VAR_GLOBAL
	/// instance array of all controller instances
	g_a_pCtrlInst: ARRAY[0..E_CtrlId.E_CtrlIdMax] OF POINTER TO fb_CtrlBase;
	/// common interface array of all controllers (main use for PLC)
	g_a_pCtrlCIf: ARRAY[0..E_CtrlId.E_CtrlIdMax] OF POINTER TO T_Ctrl_CIf;
	/// common access variabel for UI
	g_p_fbAlm_Man: POINTER TO FB_Alm_Man;
	/// Global array for function with different childs in faster cycles
	g_a_pFunRFD: ARRAY[0..9] OF POINTER TO FB_RFR;
	/// For StartUp order
	g_uinStartProzess: UINT;
	/// Count of Task Classes
	c_uinCntTaskClass: UINT := 3;
END_VAR

(* stored: Version 1.1.0.1, ProductVersion 3.1.0.23
   GVL Global: Id {c27aced4-be9c-4dab-babe-a5494623c001} *)
